// TIA Portal V20 export
FUNCTION_BLOCK "FB_FixtureBlowing"   // FB68, SCL
{ S7_Optimized_Access := 'TRUE' }
// stored: AutoNumber false, MemoryReserve 100, SetENOAutomatically false
   VAR_INPUT
      iStartSeqCond : Bool;   // Start Sequence Conditions
      iJobReq : Bool;   // Job Request - From Main
      iFixtureOpened : Bool;
      iAxisV_FixtBlowingPos : Bool;
      iAxisV_FixtBlowingPosSetPoint : LReal;
      iAxisW_FixtSafePos : Bool;
      iAxisW_FixtSafePosSetPoint : LReal;
      iAxisW_FixtBlowPos : Bool;
      iAxisW_FixtBlowPosSetPoint : LReal;
      iAxisV_Moving : Bool;   // Shuttle is moving
      iAxisV_InPos : Bool;
      iAxisW_Moving { ExternalAccessible := 'False'; ExternalVisible := 'False'; ExternalWritable := 'False'} : Bool;   // Shuttle is moving
      iAxisW_InPos : Bool;
      iBlowingTime : Time;
      iPLC_DateAndTime : DTL;
      iStepPause : Bool;
   END_VAR
   VAR_OUTPUT
      oFixtureOpenReq : Bool;
      oAxisV_StartReq : Bool;
      oAxisV_PosSetPoint : Real;
      oAxisW_StartReq : Bool;
      oAxisW_PosSetPoint : Real;
      oBlowingReq : Bool;
   END_VAR
   VAR
      sCurrent_Step_NB : Int;   // Active Step Number
      sCheck_Step_Condition : Bool;
      sOneStepForward : Bool;
      sRTOneStepForward : R_TRIG;
      sOneStepMode { S7_SetPoint := 'True'} : Bool;
      sStepForward : Bool;
      sInterface : "UDT_SequenceInterface";
      sFixtureOpenReq { S7_SetPoint := 'True'} : Bool;
      sAxisV_StartReq : Bool;
      sAxisV_PosSetPoint : Real;
      sAxisW_StartReq : Bool;
      sAxisW_PosSetPoint : Real;
      sBlowingReq : Bool;   // Drilled Part To Unload - From FB_Position
      sBlowingTimerStart : Bool;
      sBlowingTimer : TP_TIME;
      sFT_BlowingTimer { S7_SetPoint := 'True'} : F_TRIG;
      sTimerFixtureOpened : TON_TIME;
      sHistory : Struct
         Activation : Bool;
         Steps : Array[0..99] of Int;
         Date_Time : Array[0..99] of DTL;
      END_STRUCT;
      StepText : "FB_GetTextErrorCode";
   END_VAR
   VAR_TEMP
      tIndex : Int;   // Index
   END_VAR
   VAR CONSTANT
      S00_INIT : Int := 0;
      S10_CHECK_FIXTURE_BLOW_OPTION : Int := 10;
      S20_AXIS_W_TO_FIXTURE_SAFE_POS_START_REQ : Int := 20;
      S30_AXIS_W_TO_FIXTURE_SAFE_POS_REACHED : Int := 30;
      S40_AXIS_V_TO_FIXTURE_BLOW_POS_START_REQ : Int := 40;
      S50_AXIS_V_TO_FIXTURE_BLOW_POS_REACHED : Int := 50;
      S60_OPEN_FIXTURE : Int := 60;
      S70_AXIS_W_TO_FIXTURE_BLOW_POS_START_REQ : Int := 70;
      S80_AXIS_W_TO_FIXTURE_BLOW_POS_REACHED : Int := 80;
      S90_BLOWING_TIMER_START_REQ : Int := 90;
      S100_AXIS_W_TO_FIXTURE_SAFE_POS_START_REQ : Int := 100;
      S110_AXIS_W_TO_FIXTURE_SAFE_POS_REACHED : Int := 110;
      S195_JOB_DONE : Int := 195;
   END_VAR
   // StepText.sCode_error[0].ErrorCode := 0;
   // StepText.sCode_error[1].ErrorCode := 10;
   // StepText.sCode_error[2].ErrorCode := 20;
   // StepText.sCode_error[3].ErrorCode := 30;
   // StepText.sCode_error[4].ErrorCode := 40;
   // StepText.sCode_error[5].ErrorCode := 50;
   // StepText.sCode_error[6].ErrorCode := 60;
   // StepText.sCode_error[7].ErrorCode := 70;
   // StepText.sCode_error[8].ErrorCode := 80;
   // StepText.sCode_error[9].ErrorCode := 90;
   // StepText.sCode_error[10].ErrorCode := 95;
BEGIN
   REGION Description header 
       //==================================================================================
       // POSALUX Swiss SA / (C) Copyright 2026
       //----------------------------------------------------------------------------------
       // Title: FB_FixtureBlowing
       // Comment/Function: 
       // Author: Fabien WALDT
       // Engineering: TIA Portal v20
       //----------------------------------------------------------------------------------
       // Change log table:
       // Version  | Date     | Expert in charge | Changes applied
       // ---------|----------|------------------|-----------------------------------------
       // 00.00.01 | 20260122 | WFA              | First released version
       // =================================================================================
   END_REGION

   REGION Define condition to start
       IF #iStartSeqCond THEN
           #sInterface.SequenceReleased := TRUE;
       ELSE
           // Standard sequencer controls
           #sInterface.SequenceReleased := FALSE;
           #sCurrent_Step_NB := #S00_INIT;
           #sInterface.SequenceRun := FALSE;
           #sInterface.JobDone := FALSE;
           #sCheck_Step_Condition := FALSE;

           // Dedicated sequencer controls
           #sAxisV_StartReq := FALSE;
           #sAxisV_PosSetPoint := 0.0;
           #sAxisW_StartReq := FALSE;
           #sAxisW_PosSetPoint := 0.0;
           #sFixtureOpenReq := FALSE;
           #sBlowingReq := FALSE;
           #sBlowingTimerStart := FALSE;

           // Add specifics controls 
       END_IF;

       // Reset interface error
       IF #sInterface.Reset THEN
           #sInterface.Error := FALSE;
       END_IF;

       // Reset start when axis in position
       IF #iAxisV_InPos THEN
           #sAxisV_StartReq := FALSE;
       END_IF;
       IF #iAxisW_InPos THEN
           #sAxisW_StartReq := FALSE;
       END_IF;

       // One step forward
       #sRTOneStepForward.CLK := #sOneStepForward;
       #sRTOneStepForward();
       #sStepForward := (NOT #sOneStepMode OR (#sOneStepMode AND #sRTOneStepForward.Q)) AND NOT #iStepPause;
       #sOneStepForward := FALSE;

       // Blowing Timer
       #sBlowingTimer(IN := #sBlowingTimerStart,
                      PT := #iBlowingTime);

       #sFT_BlowingTimer(CLK := #sBlowingTimer.Q);

       #sBlowingReq := #sBlowingTimer.Q
       OR #sCurrent_Step_NB = 70
       OR #sCurrent_Step_NB = 80;
       // Action only true in dedicated steps
       #sFixtureOpenReq := FALSE;
       #sBlowingTimerStart := FALSE;

       // Step Timer
       #sTimerFixtureOpened(IN := #sCurrent_Step_NB = 60 AND #iFixtureOpened,
                            PT := T#1000ms);
   END_REGION

   REGION Sequence Function
       CASE #sCurrent_Step_NB OF
           #S00_INIT:
               REGION S00 INIT
                   #sCheck_Step_Condition := TRUE;
               END_REGION
           #S10_CHECK_FIXTURE_BLOW_OPTION:
               REGION S10_CHECK_FIXTURE_BLOW_OPTION
                   #sCheck_Step_Condition := TRUE;
               END_REGION
           #S20_AXIS_W_TO_FIXTURE_SAFE_POS_START_REQ:
               REGION S20_AXIS_W_TO_FIXTURE_SAFE_POS_START_REQ
                   #sAxisW_StartReq := NOT #iAxisW_FixtSafePos;
                   #sAxisW_PosSetPoint := LREAL_TO_REAL(#iAxisW_FixtSafePosSetPoint);
                   #sCheck_Step_Condition := TRUE;
               END_REGION
           #S30_AXIS_W_TO_FIXTURE_SAFE_POS_REACHED:
               REGION S30_AXIS_W_TO_FIXTURE_SAFE_POS_REACHED
                   #sCheck_Step_Condition := TRUE;
               END_REGION
           #S40_AXIS_V_TO_FIXTURE_BLOW_POS_START_REQ:
               REGION S40_AXIS_V_TO_FIXTURE_BLOW_POS_START_REQ
                   #sAxisV_StartReq := NOT #iAxisV_FixtBlowingPos;
                   #sAxisV_PosSetPoint := LREAL_TO_REAL(#iAxisV_FixtBlowingPosSetPoint);
                   #sCheck_Step_Condition := TRUE;
               END_REGION
           #S50_AXIS_V_TO_FIXTURE_BLOW_POS_REACHED:
               REGION S50_AXIS_V_TO_FIXTURE_BLOW_POS_REACHED
                   #sCheck_Step_Condition := TRUE;
               END_REGION
           #S60_OPEN_FIXTURE:
               REGION S60_OPEN_FIXTURE
                   #sFixtureOpenReq := TRUE;
                   IF #sTimerFixtureOpened.Q THEN
                       #sCheck_Step_Condition := TRUE;
                   END_IF;
               END_REGION
           #S70_AXIS_W_TO_FIXTURE_BLOW_POS_START_REQ:
               REGION S70_AXIS_W_TO_FIXTURE_BLOW_POS_START_REQ
                   #sAxisW_StartReq := NOT #iAxisW_FixtBlowPos;
                   #sAxisW_PosSetPoint := LREAL_TO_REAL(#iAxisW_FixtBlowPosSetPoint);
                   #sCheck_Step_Condition := TRUE;
               END_REGION
           #S80_AXIS_W_TO_FIXTURE_BLOW_POS_REACHED:
               REGION S80_AXIS_W_TO_FIXTURE_BLOW_POS_REACHED
                   #sCheck_Step_Condition := TRUE;
               END_REGION
           #S90_BLOWING_TIMER_START_REQ:
               REGION S90_BLOWING_TIMER_START_REQ
                   #sBlowingTimerStart := TRUE;
                   #sCheck_Step_Condition := TRUE;
               END_REGION
           #S100_AXIS_W_TO_FIXTURE_SAFE_POS_START_REQ:
               REGION S100_AXIS_W_TO_FIXTURE_SAFE_POS_START_REQ
                   #sAxisW_StartReq := NOT #iAxisW_FixtSafePos;
                   #sAxisW_PosSetPoint := LREAL_TO_REAL(#iAxisW_FixtSafePosSetPoint);
                   #sCheck_Step_Condition := TRUE;
               END_REGION
           #S110_AXIS_W_TO_FIXTURE_SAFE_POS_REACHED:
               REGION S110_AXIS_W_TO_FIXTURE_SAFE_POS_REACHED
                   #sCheck_Step_Condition := TRUE;
               END_REGION
           #S195_JOB_DONE:
               REGION S195_JOB_DONE
                   #sInterface.JobDone := TRUE;
                   #sCheck_Step_Condition := TRUE;
               END_REGION
           ELSE:
               #sInterface.Error := TRUE;
       END_CASE;
   END_REGION

   REGION Sequence Next Step Condition
       IF #sCheck_Step_Condition THEN
           CASE #sCurrent_Step_NB OF
               #S00_INIT:
                   REGION S00_INIT
                       IF #sInterface.SequenceReleased AND #iJobReq THEN
                           #sCurrent_Step_NB := #S10_CHECK_FIXTURE_BLOW_OPTION;
                           #sInterface.SequenceRun := TRUE;
                           #sCheck_Step_Condition := FALSE;
                       ELSE
                           #sInterface.SequenceRun := FALSE;
                       END_IF;
                   END_REGION
               #S10_CHECK_FIXTURE_BLOW_OPTION:
                   REGION S10_CHECK_FIXTURE_UNLOAD_OPTION
                       IF #sInterface.SequenceReleased AND #sStepForward AND NOT "DB_LoaderOptions".Fixture.BlowingDisabled  THEN
                           #sCurrent_Step_NB := #S20_AXIS_W_TO_FIXTURE_SAFE_POS_START_REQ;
                           #sCheck_Step_Condition := FALSE;
                       ELSIF #sInterface.SequenceReleased AND #sStepForward AND "DB_LoaderOptions".Fixture.BlowingDisabled THEN
                           #sCurrent_Step_NB := #S195_JOB_DONE;
                           #sCheck_Step_Condition := FALSE;
                       END_IF;
                   END_REGION
               #S20_AXIS_W_TO_FIXTURE_SAFE_POS_START_REQ:
                   REGION S20_AXIS_W_TO_FIXTURE_SAFE_POS_START_REQ
                       IF #sInterface.SequenceReleased AND #sStepForward AND (#iAxisW_Moving OR #iAxisW_FixtSafePos) THEN
                           #sCurrent_Step_NB := #S30_AXIS_W_TO_FIXTURE_SAFE_POS_REACHED;
                           #sCheck_Step_Condition := FALSE;
                       END_IF;
                   END_REGION
               #S30_AXIS_W_TO_FIXTURE_SAFE_POS_REACHED:
                   REGION S30_AXIS_W_TO_FIXTURE_SAFE_POS_REACHED
                       IF #sInterface.SequenceReleased AND #sStepForward AND NOT #sAxisW_StartReq AND #iAxisW_FixtSafePos THEN
                           #sCurrent_Step_NB := #S40_AXIS_V_TO_FIXTURE_BLOW_POS_START_REQ;
                           #sCheck_Step_Condition := FALSE;
                       END_IF;
                   END_REGION
               #S40_AXIS_V_TO_FIXTURE_BLOW_POS_START_REQ:
                   REGION S40_AXIS_V_TO_FIXTURE_BLOW_POS_START_REQ
                       IF #sInterface.SequenceReleased AND #sStepForward AND (#iAxisV_Moving OR #iAxisV_FixtBlowingPos) THEN
                           #sCurrent_Step_NB := #S50_AXIS_V_TO_FIXTURE_BLOW_POS_REACHED;
                           #sCheck_Step_Condition := FALSE;
                       END_IF;
                   END_REGION
               #S50_AXIS_V_TO_FIXTURE_BLOW_POS_REACHED:
                   REGION S50_AXIS_V_TO_FIXTURE_BLOW_POS_REACHED
                       IF #sInterface.SequenceReleased AND #sStepForward AND NOT #sAxisV_StartReq AND #iAxisV_FixtBlowingPos THEN
                           #sCurrent_Step_NB := #S60_OPEN_FIXTURE;
                           #sCheck_Step_Condition := FALSE;
                       END_IF;
                   END_REGION
               #S60_OPEN_FIXTURE:
                   REGION S60_OPEN_FIXTURE
                       IF #sInterface.SequenceReleased AND #sStepForward AND #iFixtureOpened THEN
                           #sCurrent_Step_NB := #S70_AXIS_W_TO_FIXTURE_BLOW_POS_START_REQ;
                           #sCheck_Step_Condition := FALSE;
                       END_IF;
                   END_REGION
               #S70_AXIS_W_TO_FIXTURE_BLOW_POS_START_REQ:
                   REGION S70_AXIS_W_TO_FIXTURE_BLOW_POS_START_REQ
                       IF #sInterface.SequenceReleased AND #sStepForward AND (#iAxisW_Moving OR #iAxisW_FixtBlowPos) THEN
                           #sCurrent_Step_NB := #S80_AXIS_W_TO_FIXTURE_BLOW_POS_REACHED;
                           #sCheck_Step_Condition := FALSE;
                       END_IF;
                   END_REGION
               #S80_AXIS_W_TO_FIXTURE_BLOW_POS_REACHED:
                   REGION S80_AXIS_W_TO_FIXTURE_BLOW_POS_REACHED
                       IF #sInterface.SequenceReleased AND #sStepForward AND NOT #sAxisW_StartReq AND #iAxisW_FixtBlowPos THEN
                           #sCurrent_Step_NB := #S90_BLOWING_TIMER_START_REQ;
                           #sCheck_Step_Condition := FALSE;
                       END_IF;
                   END_REGION
               #S90_BLOWING_TIMER_START_REQ:
                   REGION S90_BLOWING_TIMER_START_REQ
                       IF #sInterface.SequenceReleased AND #sStepForward AND #sFT_BlowingTimer.Q THEN
                           #sCurrent_Step_NB := #S100_AXIS_W_TO_FIXTURE_SAFE_POS_START_REQ;
                           #sCheck_Step_Condition := FALSE;
                       END_IF;
                   END_REGION
               #S100_AXIS_W_TO_FIXTURE_SAFE_POS_START_REQ:
                   REGION S100_AXIS_W_TO_FIXTURE_SAFE_POS_START_REQ
                       IF #sInterface.SequenceReleased AND #sStepForward AND (#iAxisW_Moving OR #iAxisW_FixtSafePos) THEN
                           #sCurrent_Step_NB := #S110_AXIS_W_TO_FIXTURE_SAFE_POS_REACHED;
                           #sCheck_Step_Condition := FALSE;
                       END_IF;
                   END_REGION
               #S110_AXIS_W_TO_FIXTURE_SAFE_POS_REACHED:
                   REGION S110_AXIS_W_TO_FIXTURE_SAFE_POS_REACHED
                       IF #sInterface.SequenceReleased AND #sStepForward AND NOT #sAxisW_StartReq AND #iAxisW_FixtSafePos THEN
                           #sCurrent_Step_NB := #S195_JOB_DONE;
                           #sCheck_Step_Condition := FALSE;
                       END_IF;
                   END_REGION
               #S195_JOB_DONE:
                   REGION S195_JOB_DONE
                       IF NOT #iJobReq THEN
                           #sCurrent_Step_NB := #S00_INIT;
                           #sCheck_Step_Condition := FALSE;
                           #sInterface.JobDone := FALSE;
                       END_IF;
                   END_REGION
               ELSE
                   #sInterface.Error := TRUE;
           END_CASE;
       END_IF;
   END_REGION

   REGION Outputs Update
       #oAxisV_StartReq := #sAxisV_StartReq;
       #oAxisV_PosSetPoint := #sAxisV_PosSetPoint;
       #oAxisW_StartReq := #sAxisW_StartReq;
       #oAxisW_PosSetPoint := #sAxisW_PosSetPoint;
       #oFixtureOpenReq := #sFixtureOpenReq;
       #oBlowingReq := #sBlowingReq;
   END_REGION

   REGION Steps - Date and Time History
       IF #sHistory.Activation THEN
           IF #sHistory.Steps[0] <> #sCurrent_Step_NB THEN
               FOR #tIndex := 98 TO 0 BY -1 DO
                   #sHistory.Steps[#tIndex + 1] := #sHistory.Steps[#tIndex];
                   #sHistory.Date_Time[#tIndex + 1] := #sHistory.Date_Time[#tIndex];
               END_FOR;
               #sHistory.Steps[0] := #sCurrent_Step_NB;
               #sHistory.Date_Time[0] := #iPLC_DateAndTime;
           END_IF;
       END_IF;
   END_REGION

   REGION Steps Text
       #StepText(iErrorCode := #sCurrent_Step_NB,
                 oErrorText => #StepText.oErrorText);
   END_REGION
END_FUNCTION_BLOCK
